// TIA Portal project "Aprenda a Programar CLP do ZERO - André Terra - CLP Fácil" (V15.1)
// Melhorias implementadas no código original das vídeos aulas bonus do curso "Aprenda a Simulação - "Programar CLP do ZERO" do André Terra - CLP Fácil - https://www.clpfacil.com.br

(* hardware
DEVICE "S7-1200 station_1"  S7-1200 Station
   slot 0: "Rack_0"  S7-1200 Rack  Rack  V1.0
   slot 1: "PLC MAIN"  CPU 1215C DC/DC/DC  6ES7 215-1AG40-0XB0  V4.2
*)

// ===== PLC "PLC MAIN"  CPU 1215C DC/DC/DC =====

VAR_GLOBAL   // PLC tag table "Default tag table"
   ""Botão Liga B1"" AT %I0.0 : Bool;
   ""Botão Desliga B2"" AT %I0.1 : Bool;
   ""Sensor S1"" AT %I0.2 : Bool;
   ""Sensor S2"" AT %I0.3 : Bool;
   ""Sensor S3"" AT %I0.4 : Bool;
   ""Sensor S4"" AT %I0.5 : Bool;
   ""Motor M1"" AT %Q0.0 : Bool;
   ""Motor M2"" AT %Q0.1 : Bool;
   ""Cilindro C1"" AT %Q0.2 : Bool;
END_VAR